TEXTLIST TextList_SwapInfo
  1 = 'AC_STORAGE_FLUSH_RUNS'
  2 = 'AC_STORAGE_FLUSH_NEEDS_HELP'
  3 = 'AC_STORAGE_FLUSH_FINISHED'
  4 = 'AC_WHITE_INK_RUNS'
  5 = 'AC_WHITE_INK1_NEEDS_HELP'
  6 = 'AC_WHITE_INK2_NEEDS_HELP'
  7 = 'AC_WHITE_INK_FINISHED'
   = ''
END_TEXTLIST

(* stored: Version 1.1.0.1, ProductVersion 3.1.4024.11
   TextList TextList_SwapInfo: Id {18af8894-c494-408b-b553-9fbad1ee8b14} *)
